{attribute 'linkalways'} 
{attribute 'no_explicit_call' := 'This FB is a CLASS and must be accessed using methods or properties'}
{attribute 'enable_dynamic_creation'}
FUNCTION_BLOCK Node_F_VN_CopyContainer EXTENDS VisionNode
VAR
    ipSrcContainer : _ITcVnContainer;
    ipDestContainer : _ITcVnContainer;
    hrPrev : _HRESULT(S_OK);
	hresult : _HRESULT(S_OK);
END_VAR

METHOD PUBLIC  Clone : I_Node
VAR
	pNode : POINTER TO Node_F_VN_CopyContainer;
END_VAR
pNode := __NEW(Node_F_VN_CopyContainer);
Clone := pNode^;
END_METHOD

METHOD FB_init : BOOL
VAR_INPUT
	bInitRetains : BOOL; // if TRUE, the retain variables are initialized (warm start / cold start)
	bInCopyCode : BOOL;  // if TRUE, the instance afterwards gets moved into the copy code (online change)
END_VAR
AddInput('ipSrcContainer', ipSrcContainer);
AddInput('hrPrev', hrPrev);
AddOutput('ipDestContainer', ipDestContainer);
AddOutput('hresult',hresult);
END_METHOD

METHOD PROTECTED OnExecute
hresult.Value := F_VN_CopyContainer(
	ipSrcContainer := ipSrcContainer.Value,
    ipDestContainer := ipDestContainer.Value,
	hrPrev:= hrPrev.Value);
END_METHOD

METHOD PUBLIC PreExecutionCheck
VAR_INPUT
	Check : I_PreExecutionChecks;
END_VAR
Check.IsTrue(ipSrcContainer.IsValid, 'ipSrcContainer must be a valid container');
END_METHOD

END_FUNCTION_BLOCK

(* stored: Version 1.1.0.1, ProductVersion 3.1.4024.13
   POU Node_F_VN_CopyContainer: Id {0b3ad5a2-3161-06bd-369a-7c34471b53aa}, SpecialFunc None
   Folder Constructor: Id {343c903e-da0c-072c-3535-5d85636744f5}
   Method Clone: Id {7c972433-7291-0646-0eb5-dde4d08ae7d8}
   Method FB_init: Id {2341778e-9c73-093a-2c3d-e16547623d85}
   Method OnExecute: Id {8b2d960b-9b1d-06e2-15a3-79caab43f51b}
   Method PreExecutionCheck: Id {23de2276-cf7f-0cdf-2abd-f1ac9869ca35} *)
